FUNCTION_BLOCK SP5_INTERFACE
  {SET_ATTRIBUTE(OpcUa, SERVICE)}
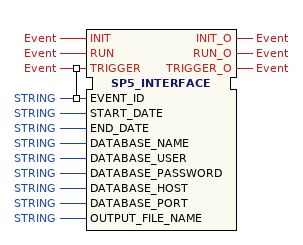
  EVENT_INPUT
    INIT;
    RUN;
    TRIGGER WITH EVENT_ID;
  END_EVENT
  EVENT_OUTPUT
    INIT_O;
    RUN_O;
    TRIGGER_O;
  END_EVENT
  VAR_INPUT
    EVENT_ID : STRING; {SET_ATTRIBUTE(OpcUa, Variable)}
    START_DATE : STRING; {SET_ATTRIBUTE(OpcUa, Constant)}
    END_DATE : STRING; {SET_ATTRIBUTE(OpcUa, Constant)}
    DATABASE_NAME : STRING; {SET_ATTRIBUTE(OpcUa, Constant)}
    DATABASE_USER  : STRING; {SET_ATTRIBUTE(OpcUa, Constant)}
    DATABASE_PASSWORD : STRING; {SET_ATTRIBUTE(OpcUa, Constant)}
    DATABASE_HOST : STRING; {SET_ATTRIBUTE(OpcUa, Constant)}
    DATABASE_PORT : STRING; {SET_ATTRIBUTE(OpcUa, Constant)}
    OUTPUT_FILE_NAME : STRING; {SET_ATTRIBUTE(OpcUa, Constant)}
  END_VAR
END_FUNCTION_BLOCK
